(* Logix 5000 project; controller Carpenter_Meter_SCP vendor 1 type 14 code 217 rev 31.11; software revision 31.01; part 3 of 7 *)

VAR_GLOBAL   (* controller tags *)
   AI_8800 : REAL := 0.44444445;   // Meter Skid MS8800 Oil Quality BS&W (%)
   AI_8840 : REAL;   // Meter Skid MS8840 Oil Quality BS&W (%)
   alarm_co : BOOL[32];
   Alarm_horn_req : BOOL;   // Alarm Horn Request
   alarm_horn_req_tmr : TIMER := (PRE := 1000);   // Alarm Horn Request Timer
   AlwaysOff : BOOL;   // Always Off Bit
   CAR100_Flowpath : BOOL;   // Carpenter MLV CAR100 Flow Path (1=OK)
   CAR100_HB_Fail : TGE_Alarm := (Enabled := 1, AlmInputState := 1, AlmExists := 1, InAlmAct := 1, InAlmHMI := 1, DelayTimerPRE := 30.0, DelayTimerACC := 29.999, Priority := 4);   // Carpenter MLV CAR100 Heartbeat Fail Alarm
   CAR100_HB_Prev : DINT;   // MLV CAR100 Previous Heartbeat
   CAR100_High_Pressure_SD : BOOL;   // Carpenter MLV CAR100 High Pressure Shutdown Status
   Carpenter_ISD_Command : BOOL;   // Carpenter/Hereford ISD Command from OCC (Through Pawnee)
   Carpenter_Status_Pawnee : DINT[50] := ([0] := 1144740586, [2] := -1072685029);   // Carpenter Status to Pawnee
   Carpenter_to_Pawnee_OK : BOOL := 1;   // Carpenter to Pawnee Flow Path Permissive
   CC_Cust1_Flow_Permissive : BOOL := 1;   // Customer #1 (MS8800) Flow Permissive to OCC
   CC_Cust1_Hi_WIOM : BOOL;   // Customer #1 High Water % Alarm to OCC
   CC_Cust1_Pump_Running : BOOL := 1;   // Customer #1 (MS8800) Pump Running Status to OCC
   CC_Cust1_Ready : BOOL := 1;   // Customer #1 (MS8800) Ready Status to OCC
   CC_Cust1_Shutin_Timer : REAL := 30.0;   // Customer #1 Shutin Reset Time Left to OCC
   CC_Cust1_Shutin_Timer1 : DINT := 30;   // Customer #1 Shutin Reset Time Left to OCC
   CC_Cust1_WIOM_Shutin : BOOL;   // Customer #1 Shutin Due to High High Water in Oil Monitor Alarm to OCC
   CC_Cust2_Flow_Permissive : BOOL;   // Customer #2 (MS8810) Flow Permissive to OCC
   CC_Cust3_Flow_Permissive : BOOL;   // Customer #3 (MS8820) Flow Permissive to OCC
   CC_Cust4_Flow_Permissive : BOOL;   // Customer #4 (MS8830) Flow Permissive to OCC
   CC_Cust5_Flow_Permissive : BOOL := 1;   // Customer #5 (MS8840) Flow Permissive to OCC
   CC_Cust5_Pump_Running : BOOL;   // Customer #5 (MS8840) Pump Running Status to OCC
   CC_Cust5_Ready : BOOL := 1;   // Customer #5 (MS8840) Ready Status to OCC
   CC_Hererford_Flow_Path : BOOL;   // Flow Path to Hereford
   CC_HI_8800 : BOOL;   // Meter Skid MS-8800 Intrusion Deactivate Switch to OCC
   CC_HI_8840 : BOOL;   // Meter Skid MS-8840 Intrusion Deactivate Switch to OCC
   CC_MS8800_Biocide_Flow : REAL;   // Meter Skid MS-8800 Biocide Flow Rate
   CC_MS8800_Biocide_Flow_SP : REAL := 3.7771018;   // Meter Skid MS-8800 Biocide Flow Rate Setpoint
   CC_MS8800_CustPress : OCC_Analog := (scaled := 70.41581);   // Meter Skid MS-8800 Customer Inlet Pressure to OCC
   CC_MS8810_CustPress : OCC_Analog;   // Meter Skid MS-8810 Customer Inlet Pressure to OCC
   CC_MS8820_CustPress : OCC_Analog;   // Meter Skid MS-8820 Customer Inlet Pressure to OCC
   CC_MS8830_CustPress : OCC_Analog;   // Meter Skid MS-8830 Customer Inlet Pressure to OCC
   CC_MS8840_Biocide_Flow : REAL;   // Meter Skid MS-8800 Biocide Flow Rate
   CC_MS8840_Biocide_Flow_SP : REAL := 1.3565929;   // Meter Skid MS-8800 Biocide Flow Rate Setpoint
   CC_MS8840_CustPress : OCC_Analog := (scaled := 158.50713);   // Meter Skid MS-8840 Customer Inlet Pressure to OCC
   CC_OCC_HB : DINT := 12;   // Heartbeat from OCC to SCP
   CC_Pawnee_Flow_Path : BOOL := 1;   // Flow Path to Pawnee
   CC_PI_1101 : OCC_Analog;   // Station Discharge Pressure to OCC
   CC_PV_0001 : OCC_CV := (Pos := 100.0738, PosCmd := 100.0);   // PV-0001
   CC_PV_0001_Flow_SP : DINT := 1000;   // Meter Skid MS8800 Inlet Control Valve Flow Setpoint
   CC_PV_0001_Press_SP : DINT := 5;   // Meter Skid MS8800 Inlet Control Valve Press Setpoint
   CC_PV_0041 : OCC_CV := (Pos := 32.79953, PosCmd := 33.05351);   // PV-0041
   CC_PV_0041_Flow_SP : DINT := 500;   // Meter Skid MS8840 Inlet Control Valve Flow Setpoint
   CC_PV_0041_Press_SP : DINT := 120;   // Meter Skid MS8800 Inlet Control Valve Press Setpoint
   CC_SCP_HB : DINT := 1658;   // Heartbeat from SCP to OCC
   CC_STA_Stop : BOOL;   // Station Stop Request Command from OCC
   CC_XA_0020A : BOOL;   // SCP Main Panel 24VDC Fail to OCC
   CC_XA_0021A : BOOL;   // FGP Main Panel 24VDC Fail to OCC
   CC_XI_0001 : BOOL;   // QA Building Intrusion Deactivate Switch to OCC
   CC_XI_0001A : BOOL := 1;   // QA Building Intrusion Switch to OCC
   CC_XI_0011A : BOOL := 1;   // PDC Building Intrusion Switch to OCC
   CC_XI_0011B : BOOL := 1;   // PDC Building Intrusion Deactivate Switch to OCC
   CC_XI_0020 : BOOL;   // SCP Main PLC 24VDC Failure to OCC
   CC_XI_0021 : BOOL;   // FGP Main PLC 24VDC Failure to OCC
   CC_XI_8800 : BOOL;   // Meter Skid MS-8800 Intrusion Switch to OCC
   CC_XI_8800A : BOOL;   // MS8800 SCP 24VDC Failure to OCC
   CC_XI_8800B : BOOL;   // MS8800 FGP 24VDC Failure to OCC
   CC_XI_8840 : BOOL;   // Meter Skid MS-8840 Intrusion Switch to OCC
   CC_XI_8840A : BOOL;   // MS8840 SCP 24VDC Failure to OCC
   CC_XI_8840B : BOOL;   // MS8840 FGP 24VDC Failure to OCC
   CC_YI_6000 : BOOL;   // UPS-6000 Utility Power Loss to OCC
   CC_YI_6001 : BOOL;   // UPS-6000 Fault
   CC_ZI_1100A : BOOL;   // Pig Launched Pig Sig to OCC
   CC_ZI_1100B : BOOL;   // Pig Station Depart Pig Sig to OCC
   CCS_AI_0001 : OCC_Analog := (scaled := 0.024822354);   // QA Building Gas Detector to OCC (AIT-0001)
   CCS_AI_8800A : OCC_Analog := (scaled := 0.18368065);   // Meter Skid MS-8800 Gas Detector #1 (AIT-8800A)
   CCS_AI_8800B : OCC_Analog := (scaled := 0.21929741);   // Meter Skid MS-8800 Gas Detector #2 (AIT-8800B)
   CCS_AI_8840A : OCC_Analog := (scaled := 0.25642216);   // Meter Skid MS-8840 Gas Detector #1 (AIT-8840A)
   CCS_AI_8840B : OCC_Analog := (scaled := 0.22641718);   // Meter Skid MS-8840 Gas Detector #2 (AIT-8840B)
   CCS_ESD_Active : BOOL;   // Station ESD Active to OCC
   CCS_ESD_OCC : BOOL;   // Station ESD Command from OCC
   CCS_FGP_Deactivate : BOOL;   // Fire and Gas Deactivated Status to OCC
   CCS_HI_0011A : BOOL;   // PDC ESD Pushbutton to OCC
   CCS_HI_0017 : BOOL;   // PDC Building PLC Panel ESD Pushbutton to OCC
   CCS_HI_0112A : BOOL;   // QA Building ESD Pushbutton #1 to OCC
   CCS_HI_0112B : BOOL;   // QA Building ESD Pushbutton #2 to OCC
   CCS_HI_0113 : BOOL;   // South Gate ESD Pushbutton to OCC
   CCS_HI_0114 : BOOL;   // North Gate ESD Pushbutton to OCC
   CCS_HI_0115 : BOOL;   // Site ESD Pushbutton #3 to OCC - Currently Unused
   CCS_HI_8800A : BOOL;   // Meter Skid MS-8800 ESD Pushbutton #1 to OCC
   CCS_HI_8800B : BOOL;   // Meter Skid MS-8800 ESD Pushbutton #2 to OCC
   CCS_HI_8840A : BOOL;   // Meter Skid MS-8840 ESD Pushbutton #1 to OCC
   CCS_HI_8840B : BOOL;   // Meter Skid MS-8840 ESD Pushbutton #1 to OCC
   CCS_LAH_3000 : BOOL;   // Sump Tank TU-3000 Leak Detection Switch to OCC
   CCS_LAH_3000_inhibit : BOOL;   // Sump Tank TU-3000 Leak Detection Switch Inhibited to OCC
   CCS_LAH_3100 : BOOL;   // Sump Tank TU-3100 Leak Detection Switch to OCC
   CCS_LAH_3100_inhibit : BOOL;   // Sump Tank TU-3100 Leak Detection Switch Inhibited to OCC
   CCS_LAHH_3000 : BOOL;   // Sump Tank TU-3000 HiHi Level Switch to OCC
   CCS_LAHH_3000_inhibit : BOOL;   // Sump Tank TU-3000 HiHi Level Switch Inhibited to OCC
   CCS_LAHH_3100 : BOOL;   // Sump Tank TU-3100 HiHi Level Switch to OCC
   CCS_LAHH_3100_inhibit : BOOL;   // Sump Tank TU-3100 HiHi Level Switch inhibited to OCC
   CCS_LI_3000 : OCC_Analog;   // Sump Tank TU-3000 Level to OCC
   CCS_LI_3100 : OCC_Analog := (scaled := 27.158325);   // Sump Tank TU-3000 Level to OCC
   CCS_TI_8010 : OCC_Analog := (scaled := -50.0);   // PDC Building Temperature (TIT-8010)
   CCS_XI_0029A : BOOL;   // QA Building Smoke Detector #1 to OCC
   CCS_XI_0029A_Inhibit : BOOL;   // QA Building Smoke Detector #1 Inhibit to OCC
   CCS_XI_0029B : BOOL;   // QA Building Smoke Detector #2 to OCC
   CCS_XI_0029B_Inhibit : BOOL;   // QA Building Smoke Detector #2 Inhibit to OCC
   CCS_XV_0001 : BaseVLVLiquid := (chg_tmr.PRE := 180000, Close_Req_Tmr.PRE := 20000, Expected := 1, Last_Pos := 1, Open_Req_Tmr.PRE := 20000, Opn_Sts := 1, Startup_bit := 1, Startup_tmr.PRE := 120000, remote := 1, OOP_alm.sta_attended := 1, OOP_alm.alm_tmr_pre := 180000, status := 1);   // XV-0001 OCC
   CCS_XV_0041 : BaseVLVLiquid := (chg_tmr.PRE := 180000, Close_Req_Tmr.PRE := 20000, Expected := 1, Last_Pos := 1, Open_Req_Tmr.PRE := 20000, Opn_Sts := 1, Startup_bit := 1, Startup_tmr.PRE := 120000, remote := 1, OOP_alm.sta_attended := 1, OOP_alm.alm_tmr_pre := 180000, status := 1);   // XV-0041 OCC
   CCS_XV_1100 : BaseVLVLiquid := (chg_tmr.PRE := 180000, Close_Req_Tmr.PRE := 20000, Cls_Sts := 1, Open_Req_Tmr.PRE := 20000, Startup_bit := 1, Startup_tmr.PRE := 120000, remote := 1, OOP_alm.sta_attended := 1, OOP_alm.alm_tmr_pre := 180000, status := 2);   // XV-1100 OCC
   CCS_XV_1101 : BaseVLVLiquid := (chg_tmr.PRE := 180000, Close_Req_Tmr.PRE := 20000, Expected := 1, Last_Pos := 1, Open_Req_Tmr.PRE := 20000, Opn_Sts := 1, Startup_bit := 1, Startup_tmr.PRE := 120000, remote := 1, OOP_alm.sta_attended := 1, OOP_alm.alm_tmr_pre := 180000, status := 1);   // XV-1101 OCC
   CCS_YI_0022A : BOOL;   // PDC Smoke Detector to OCC
   CCS_YI_0022A_Inhibit : BOOL;   // PDC Smoke Detector Inhibit to OCC
   cmd_reset_tmr : TIMER[8] := ([0].PRE := 2000, [1].PRE := 2000, [2].PRE := 2000);   // General Use HMI Command Reset Timer
   Cust1_WIOM_Alarm : BOOL;   // Customer 1 WIOM Alarm
   Cust1_WIOM_High_Tmr : TIMER := (PRE := 900000, ACC := 82173, EN := 1, TT := 1);   // Customer 1 Water in Oil Monitor Alarm Timer
   Cust1_WIOM_Reset : BOOL;   // Customer 1 WIOM Reset Lockout from HMI
   Cust1_WIOM_Reset_Tmr : TIMER := (PRE := 1800000);   // Customer 1 Reset Timer for a WIOM Shutin
   Customer1_Flowpath_OK : BOOL := 1;   // Customer #1 Flowpath Permissive (1 = OK)
   Customer1_Pump_Status : BOOL := 1;   // Customer #1 Pump Running Status
   Customer1_Ready_Status : BOOL := 1;   // Customer #1 Ready Status
   Customer2_Flowpath_OK : BOOL;   // Customer #1 Flowpath Permissive (1 = OK)
   Customer3_Flowpath_OK : BOOL;   // Customer #3 Flowpath Permissive (1 = OK)
   Customer4_Flowpath_OK : BOOL;   // Customer #4 Flowpath Permissive (1 = OK)
   Customer4_HB : DINT;
   Customer5_Flowpath_OK : BOOL := 1;   // Customer #5 Flowpath Permissive (1 = OK)
   Customer5_Ready_Status : BOOL := 1;   // Customer #4 Ready Status
   DI_8800 : REAL := 35.538742;   // Meter Skid MS8800 Density (API)
   DI_8800_Batch : REAL := 35.5;   // Meter Skid MS8800 Current Batch Density (API)
   DI_8800_Live : REAL := 36.08286;   // Meter Skid MS8800 Live Observed Density (API)
   DI_8800_PrevBatch : REAL := 35.3;   // Meter Skid MS8800 Previous Batch Density (API)
   DI_8840 : REAL := 34.859913;   // Meter Skid MS8840 Density (API)
   DI_8840_Batch : REAL := 34.9;   // Meter Skid MS8840 Current Batch Density (API)
   DI_8840_Live : REAL := 34.490906;   // Meter Skid MS8840 Indicated Volume (Raw) (BBL/HR)
   DI_8840_PrevBatch : REAL := 35.2;   // Meter Skid MS8840 Previous Batch Density (API)
   fgp_deactivate_keysw : BOOL;   // Fire and Gas System Deactivated through Key Switch
   FGP_ESD : TGE_Alarm := (Enabled := 1, AlmExists := 1);   // ESD Shutdown from FGP (HS-0020A)
   FGP_Fire_Det : TGE_Alarm := (Enabled := 1, AlmExists := 1);   // Fire Shutdown from FGP (YSHH-0022)
   FGP_Gas_Det : TGE_Alarm := (Enabled := 1, AlmExists := 1);   // Hi Gas Shutdown from FGP (ASHH-0021)
   FGP_HB_Fail_Alm : TGE_Alarm := (Enabled := 1, AlmExists := 1);   // FGP Heartbeat Failure Alarm
   fgp_panel_reset : BOOL;   // FGP Panel Reset Pushbutton
   FGP_Produced : BasProdCons := (integer[1] := 6, integer[2] := 5, integer[3] := 5, integer[7] := 5, float[30] := 21829.0);   // FGP Produced Data
   FGP_SCADA : BasProdCons := (bit[31] := 1, bit[34] := 1, float[0] := 0.15720427, float[1] := 0.20538867, float[2] := 0.20030737, float[3] := 0.27327836, float[4] := 0.22177398, float[5] := -50.0);
   FI_8800 : REAL := 749.4378;   // Meter Skid MS-8800 Flow Rate in GSV from EFM
   FI_8800_Batch : REAL := 122.67;   // Meter Skid MS8800 Current Batch Volume in GSV (BBL)
   FI_8800_PrevBatch : REAL := 15693.27;   // Meter Skid MS8800 Pervious Batch Volume in GSV (BBL)
   FI_8800_Raw : REAL := 739.0667;   // Meter Skid MS8800 Indicated Volume (Raw) (BBL/HR)
   FI_8840 : REAL := 364.02893;   // Meter Skid MS-8840 Flow Rate from EFM
   FI_8840_Batch : REAL := 43.56;   // Meter Skid MS8840 Current Batch Volume in GSV (BBL)
   FI_8840_PrevBatch : REAL := 4837.04;   // Meter Skid MS8840 Pervious Batch Volume in GSV (BBL)
   FI_8840_Raw : REAL := 371.8956;   // Meter Skid MS8840 Indicated Volume (Raw) (BBL/HR)
   FQI_8800_DriveGain : REAL := 3.6537004;   // Meter Skid MS8800 Drive Gain (%)
   FQI_8800_Factor : REAL;   // Meter Skid MS8800 Meter Factor
   FQI_8800_LastMonth : REAL;   // Meter Skid MS8800 Gross Standard Volume Last Month (BBL)
   FQI_8800_MassFlow : REAL := 3645.5835;   // Meter Skid MS8800 Coriolis Mass Flow Rate (lb/min)
   FQI_8800_MassTotal : REAL := 774424400.0;   // Meter Skid MS8800 Coriolis Mass Totalizer (lb)
   FQI_8800_ThisMonth : REAL;   // Meter Skid MS8800 Gross Standard Volume This Month (BBL)
   FQI_8800_Today : REAL;   // Meter Skid MS8800 Gross Standard Volume Today (BBL)
   FQI_8800_Total : REAL;   // Meter Skid MS8800 Gross Standard Volume Total (BBL)
   FQI_8800_Yesterday : REAL;   // Meter Skid MS8800 Gross Standard Volume Yesterday (BBL)
   FQI_8840_DriveGain : REAL := 7.312943;   // Meter Skid MS8840 Drive Gain (%)
   FQI_8840_Factor : REAL;   // Meter Skid MS8840 Meter Factor
   FQI_8840_LastMonth : REAL;   // Meter Skid MS8840 Gross Standard Volume Last Month (BBL)
   FQI_8840_MassFlow : REAL := 1854.8619;   // Meter Skid MS8840 Coriolis Mass Flow Rate (lb/min)
   FQI_8840_MassTotal : REAL := 46132996.0;   // Meter Skid MS8840 Coriolis Mass Totalizer (lb)
   FQI_8840_ThisMonth : REAL;   // Meter Skid MS8840 Gross Standard Volume This Month (BBL)
   FQI_8840_Today : REAL;   // Meter Skid MS8840 Gross Standard Volume Today (BBL)
   FQI_8840_Total : REAL;   // Meter Skid MS8840 Gross Standard Volume Total (BBL)
   FQI_8840_Yesterday : REAL;   // Meter Skid MS8840 Gross Standard Volume Yesterday (BBL)
   hb_fail_FGP : BOOL;   // FGP Heartbeat Fail
   hb_fail_scada : BOOL;   // SCADA HB Failure
   hb_FGP : DINT := 22489;   // FGP Heartbeat
   hb_fgp_old : DINT := 22669;   // Old OCC HB for diagnostic purposes
   hb_timer_FGP : TIMER := (PRE := 600000, ACC := 15, EN := 1, TT := 1);   // FGP HB Timer
   hb_timer_scada : TIMER := (PRE := 600000, ACC := 841, EN := 1, TT := 1);   // SCADA HB Timer
   Hereford_Flowpath : BOOL := 1;   // Pawnee Terminal Flow Path (1=OK)
   Hereford_HB_Fail : TGE_Alarm := (Enabled := 1, AlmInputState := 1, AlmExists := 1, DelayTimerPRE := 30.0, DelayTimerACC := 1.527, Priority := 4);   // Hereford Heartbeat Fail Alarm
   Hereford_HB_Prev : DINT := 52;   // Hereford Previous Heartbeat
   Hereford_High_Pressure_SD : BOOL;   // Hereford High Pressure Shutdown Status
   Hereford_Msg1 : MESSAGE;
        MessageParameters(ServiceCode := 16#004c, LocalElement := Hereford_Status[0], ...)
   Hereford_OCC_HB_FAIL : BOOL;   // Pawnee High Pressure Shutdown Status
   Hereford_Status : DINT[50] := ([0] := 52, [1] := 1);   // Hereford Status Tags
   HRF100_Flowpath : BOOL := 1;   // Hereford MLV HRF100 Flow Path (1=OK)
   HRF100_HB_Fail : TGE_Alarm := (Enabled := 1, AlmInputState := 1, AlmExists := 1, DelayTimerPRE := 30.0, DelayTimerACC := 1.879);   // Hereford MLV HRF100 Heartbeat Fail Alarm
   HRF100_HB_Prev : DINT := 16;   // Hereford MLV HRF100 Previous Heartbeat
   HRF100_High_Pressure_SD : BOOL;   // Hereford MLV HRF100 High Pressure Shutdown Status
   intrusion_sys_active : BOOL;   // Intrusion System Active
   Launcher_Pig_Sig : TGE_Alarm := (Enabled := 1, AlmExists := 1);   // Launcher Pig Signal (ZS-1100A)
   Main_FGP_24VDC_Fail : TGE_Alarm := (Enabled := 1, AlmExists := 1);   // Main PLC FGP 24VDC Fail (XS-0021)
   message_timer : TIMER[10] := ([0].PRE := 5000, [0].ACC := 4855, [0].EN := 1, [0].TT := 1, [1].PRE := 2000, [1].ACC := 821, [1].EN := 1, [1].TT := 1, [2].PRE := 2000, [4].PRE := 2000);
   MLV_CAR100_Msg1 : MESSAGE;   // Carpenter MLV (CAR100) Messaging
        MessageParameters(ServiceCode := 16#004c, LocalElement := MLV_CAR100_Status[0], ...)
   MLV_CAR100_Status : DINT[50];
   MLV_HRF100_Msg1 : MESSAGE;   // Hereford MLV (HRF100) Messaging
        MessageParameters(ServiceCode := 16#004c, LocalElement := MLV_HRF100_Status[0], ...)
   MLV_HRF100_Status : DINT[50] := ([0] := 16, [1] := 1);
   mod_faultcode : DINT[10];   // PLC Module Fault Code
        [0]   // Controller Fault Code
        [1]   // SCP Main Flex I/O Fault Code
        [2]   // Meter Skid MS8800 RIO Fault Code
        [3]   // Meter Skid MS8810 RIO Fault Code
        [4]   // Meter Skid MS8820 RIO Fault Code
        [5]   // Meter Skid MS8830 RIO Fault Code
        [6]   // Meter Skid MS8840 RIO Fault Code
   mod_status : DINT[10] := ([0] := 12640, [1] := 16384, [2] := 16384, [6] := 16384, [8] := 2);   // PLC Module Status
        [0]   // Controller Module Status
        [1]   // SCP Main Flex I/O Module Status
        [2]   // Meter Skid MS8800 RIO Module Status
        [3]   // Meter Skid MS8810 RIO Module Status
        [4]   // Meter Skid MS8820 RIO Module Status
        [5]   // Meter Skid MS8830 RIO Module Status
        [6]   // Meter Skid MS8840 RIO Module Status
   MS8800_Biocide_BBL_Per_Day : REAL := 0.08833598;   // MS8800 Biocide Flow Rate in BBL/Day (Based off set target of 500PPM)
   MS8800_Biocide_Flow_Fdbk : TGE_AI_UDT := (TrendTime := 1, Raw := -3.2007636e-05, HHAlm.AlmInputState := 1, HHAlm.AlmExists := 1, HAlm.AlmInputState := 1, HAlm.AlmExists := 1, LAlm.AlmInputState := 1, LAlm.AlmExists := 1, LLAlm.AlmInputState := 1, LLAlm.AlmExists := 1, ROCNegAlm.AlmExists := 1, ROCPosAlm.AlmExists := 1, MalfAlm.AlmInputState := 1, MalfAlm.AlmExists := 1);   // Meter Skid MS-8800 Biocide Injection Rate Feedback
   MS8800_Biocide_Flow_Fdbk_AOI : TGE_AI := (Raw := -2.8205577e-05);   // Meter Skid MS-8800 Biocide Injection Rate Feedback
   MS8800_Biocide_Flow_SP : REAL := 3.7771666;   // Meter Skid MS-8800 Biocide Flow Rate Gal/Day
   MS8800_Biocide_RunReq : BOOL := 1;   // Meter Skid MS8800 Biocide Run Req
   MS8800_Cust_Press : TGE_AI_UDT := (TrendTime := 1, Avg := 70.44822, EU := 70.44822, EUMax := 1500.0, Raw := 4.7514477, RawMax := 20.0, RawMin := 4.0, Percent := 4.696548, HHAlm.AlmInputState := 1, HHAlm.AlmExists := 1, HAlm.AlmInputState := 1, HAlm.AlmExists := 1, LAlm.AlmExists := 1, LLAlm.AlmExists := 1, ROCNegAlm.AlmExists := 1, ROCPosAlm.AlmExists := 1, MalfAlm.AlmExists := 1, Average.Input := 70.44822, Average.Output := 70.44822);   // Meter Skid MS-8800 Customer Inlet Pressure (Communicated from Cust)
   MS8800_Cust_Press_AOI : TGE_AI := (Raw := 4.7514477, EU := 70.44822, Avg := 70.44822);   // Meter Skid MS-8800 Customer Inlet Pressure (Communicated from Cust)
   MS8800_Customer_Inlet_Press : AnalogAlm := (mA := 4.0, sta_attended := 1, Lo_setpt := -1.0, LoLo_setpt := -1.0, Hi_setpt := 1368.0, HiHi_setpt := 1425.0);   // Meter Skid MS8800 Customer Inlet Pressure
   MS8800_CustPress : REAL;
   MS8800_EFM_Data : REAL[50] := ([0] := 736.1332, [1] := 55.73959, [2] := 67.49643, [3] := 35.54057, [4] := 123.28, [5] := 63.0, [6] := 67.3, [7] := 35.5, [8] := 15693.27, [9] := 138.0, [10] := 65.9, [11] := 35.3, [12] := 738.34155, [13] := 36.08286, [15] := 0.44444445, [16] := 31.093464, [17] := 1.6411064, [18] := 3645.5835, [19] := 774424400.0, [20] := 3.6537004);   // MS8800 EFM Data Points
        [0]   // Live GSV Rate from MS8800 EFM
        [1]   // Live Static Pressure from MS8800 EFM
        [2]   // Live Temperature from MS8800 EFM
        [3]   // Current Batch GSV Total from MS8800 EFM
        [4]   // Current Batch FWA Static Pressure from MS8800 EFM
        [5]   // Current Batch FWA Temperature from MS8800 EFM
        [6]   // Current Batch FWA Base Density from MS8800 EFM
        [7]   // Previous Batch GSV Total from MS8800 EFM
        [8]   // Previous Batch FWA Static Pressure from MS8800 EFM
        [9]   // Previous Batch FWA Temperature from MS8800 EFM
        [10]   // Previous Batch FWA Base Density from MS8800 EFM
        [11]   // Live Indicated Volume (Raw) Rate from MS8800 EFM
        [12]   // Live Observed Density from MS8800 EFM
        [13]   // GSV Accumulator Grand Total from MS8800 EFM
        [14]   // WIOM / H20 / BSW from MS8800 EFM
        [15]   // Control Valve Position Feedback from MS8800 EFM
        [16]   // Strainer Differential from MS8800 EFM
        [17]   // Coriolis Mass Rate from MS8800 EFM
        [18]   // Coriolis Mass Totalizer from MS8800 EFM
        [19]   // Drive Gain from MS8800 EFM
        [20]   // Meter Factor from MS8800 EFM
        [21]   // Today GSV Total from MS8800 EFM
        [22]   // Yesterday GSV Total from MS8800 EFM
        [23]   // This Month GSV Total from MS8800 EFM
        [24]   // Last Month GSV Total from MS8800 EFM
   MS8800_FGP_24VDC_Fail : TGE_Alarm := (Enabled := 1, AlmExists := 1, DelayTimerPRE := 5.0, DelayTimerACC := 4.999);   // Meter Skid MS-8800 FGP 24VDC Fail (XS-8800B)
   MS8800_Flow_Control : PID := (CTL := -2147446144, EN := 1, INI := 1, OLH := 1, DVPA := 1, PVHA := 1, SP := 1000.0, KP := 0.0025, KI := 0.001, MAXS := 5000.0, DB := 7.0, SO := 100.0, MAXO := 100.0, UPD := 0.2, PV := 750.19684, ERR := 249.80316, OUT := 100.0, MAXI := 5000.0, MAXCV := 100.0, MAXTIE := 4095.0, DATA[0] := 99.99973, DATA[1] := -240.06299, DATA[2] := 750.19684, DATA[3] := 249.80316, DATA[4] := 1000.0, DATA[5] := 0.02, DATA[6] := 1.0, DATA[7] := 3.2, DATA[8] := 0.0025, DATA[9] := 0.001, DATA[11] := 0.0025, DATA[12] := 0.001, DATA[15] := 1.0, DATA[16] := 0.024420025);   // Meter Skid MS8800 Flow Rate P&ID
   MS8800_Inlet_Press : TGE_AI_UDT := (HHAlm.AlmExists := 1, HAlm.AlmExists := 1, LAlm.AlmExists := 1, LLAlm.AlmExists := 1, ROCNegAlm.AlmExists := 1, ROCPosAlm.AlmExists := 1, MalfAlm.AlmExists := 1);   // Meter Skid MS-8800 Inlet Pressure
   MS8800_Inlet_Press_AOI : TGE_AI;   // Meter Skid MS-8800 Inlet Pressure
   MS8800_Inlet_Press_Control : PID := (CTL := -2113891712, EN := 1, CA := 1, INI := 1, OLH := 1, DVPA := 1, PVHA := 1, SP := 5.0, KP := 0.2, KI := 0.05, MAXS := 1500.0, DB := 2.0, SO := 100.0, MAXO := 100.0, UPD := 0.2, PV := 70.54263, ERR := 65.54263, OUT := 100.0, MAXI := 1500.0, MAXCV := 100.0, MAXTIE := 4095.0, DATA[0] := 99.8426, DATA[1] := 75.245476, DATA[2] := 70.54263, DATA[3] := 65.54263, DATA[4] := 5.0, DATA[5] := 0.06666667, DATA[6] := 1.0, DATA[7] := 1.6, DATA[8] := 0.2, DATA[9] := 0.05, DATA[11] := 0.2, DATA[12] := 0.05, DATA[15] := 1.0, DATA[16] := 0.024420025);   // Meter Skid MS8800 Customer Inlet Pressure P&ID
   MS8800_Intrusion : IntrusionAlm := (sta_attended := 1, sw_input := 7);   // Meter Skid MS-8800 Intrusion #1 Alarm
   MS8800_OilFlow_BBL_Per_Day : REAL := 17986.508;   // Meter Skid MS-8800 Oil Flow Rate in BBL/Day
   MS8800_PCV_Pos : TGE_AI_UDT := (TrendTime := 1, Avg := 100.0739, EU := 100.0739, EUMax := 100.0, Raw := 100.0739, RawMax := 100.0, Percent := 100.0739, HHAlm.AlmInputState := 1, HHAlm.AlmExists := 1, HAlm.AlmInputState := 1, HAlm.AlmExists := 1, LAlm.AlmExists := 1, LLAlm.AlmExists := 1, ROCNegAlm.AlmExists := 1, ROCPosAlm.AlmExists := 1, MalfAlm.AlmExists := 1, Average.Input := 100.0739, Average.Output := 100.0739);   // Meter Skid MS-8800 Pressure Control Valve - Position Feedback (PCV-0001)
   MS8800_PCV_Pos_AOI : TGE_AI := (Raw := 100.07354, EU := 100.07354, Avg := 100.07354);   // Meter Skid MS-8800 Pressure Control Valve - Position Feedback (PCV-0001)
   MS8800_RIO_Fail : TGE_Alarm := (AlmInputState := 1, AlmExists := 1);   // MS8800 RIO Failure
   MS8800_WaterFlow_BBL_Per_Day : REAL := 176.67195;   // MS8800 Water Flow Rate in BBL/Day (Based off 1% oil in water)
   MS8800_WIOM_Alarm : AnalogAlm := (Input := 0.44566545, mA := 4.0, sta_attended := 1, Hi_setpt := 1.5, HiHi_setpt := 1.7, Hi_tmr_pre := 300000, HiHi_tmr_pre := 900000);   // MS8800 Water In Oil Monitor Alarm (Setpoint Dictated by Tarrif)
   MS8810_RIO_Fail : TGE_Alarm := (AlmExists := 1);   // MS8810 RIO Failure
   MS8840_Biocide_BBL_Per_Day : REAL := 0.044638067;   // MS8840 Biocide Flow Rate in BBL/Day (Based off set target of 500PPM)
   MS8840_Biocide_Flow_Fdbk : TGE_AI_UDT := (TrendTime := 1, Raw := 0.00016698558, HHAlm.AlmInputState := 1, HHAlm.AlmExists := 1, HAlm.AlmInputState := 1, HAlm.AlmExists := 1, LAlm.AlmInputState := 1, LAlm.AlmExists := 1, LLAlm.AlmInputState := 1, LLAlm.AlmExists := 1, ROCNegAlm.AlmExists := 1, ROCPosAlm.AlmExists := 1, MalfAlm.AlmInputState := 1, MalfAlm.AlmExists := 1);   // Meter Skid MS-8840 Biocide Injection Rate Feedback
   MS8840_Biocide_Flow_Fdbk_AOI : TGE_AI := (Raw := 0.00015556542);   // Meter Skid MS-8840 Biocide Injection Rate Feedback
   MS8840_Biocide_Flow_SP : REAL := 1.8475137;   // Meter Skid MS-8840 Biocide Flow Rate Gal/Day
   MS8840_Biocide_RunReq : BOOL := 1;   // Meter Skid MS8840 Biocide Run Req
   MS8840_Cust_Press : TGE_AI_UDT := (TrendTime := 1, Avg := 151.95697, EU := 151.95697, EUMax := 1650.0, Raw := 5.473522, RawMax := 20.0, RawMin := 4.0, Percent := 9.209514, HHAlm.AlmInputState := 1, HHAlm.AlmExists := 1, HAlm.AlmInputState := 1, HAlm.AlmExists := 1, LAlm.AlmExists := 1, LLAlm.AlmExists := 1, ROCNegAlm.AlmExists := 1, ROCPosAlm.AlmExists := 1, MalfAlm.AlmExists := 1, Average.Input := 151.95697, Average.Output := 151.95697);   // Meter Skid MS-8840 Customer Inlet Pressure (Communicated from Cust)
   MS8840_Cust_Press_AOI : TGE_AI := (Raw := 5.469001, EU := 151.4907, Avg := 151.4907);   // Meter Skid MS-8840 Customer Inlet Pressure (Communicated from Cust)
   MS8840_Customer_Inlet_Press : AnalogAlm := (mA := 4.0, sta_attended := 1, Lo_setpt := -1.0, LoLo_setpt := -1.0, Hi_setpt := 1368.0, HiHi_setpt := 1425.0);   // Meter Skid MS8840 Customer Inlet Pressure
   MS8840_CustPress : REAL;   // Meter Skid MS8840 Customer Inlet Pressure from Customer
   MS8840_EFM_Data : REAL[50] := ([0] := 371.9839, [1] := 110.6033, [2] := 56.4323, [3] := 34.859913, [4] := 43.56, [5] := 89.0, [6] := 56.4, [7] := 34.9, [8] := 4837.04, [9] := 124.0, [10] := 56.2, [11] := 35.2, [12] := 371.15622, [13] := 34.487686, [16] := 23.901098, [17] := 1.2, [18] := 1852.3253, [19] := 46132870.0, [20] := 7.3661847);   // MS8840 EFM Data Points
   MS8840_EFM_DINTs : DINT[10] := ([0] := 17955, [1] := 1, [2] := 144, [3] := 34, [5] := 1);   // MS8840 EFM DINT Points
        [5].1   // MS8840 EFM DINT Points
   MS8840_EFM_ReadBools : BOOL[32];   // MS8840 EFM Read Bools
   MS8840_EFM_WriteBools : BOOL[32];   // MS8840 EFM Writen Bools
   MS8840_FGP_24VDC_Fail : TGE_Alarm := (Enabled := 1, AlmExists := 1);   // Meter Skid MS-8840 FGP 24VDC Fail (XS-8840B)
   MS8840_Flow_Control : PID := (CTL := 37504, INI := 1, OLH := 1, DVPA := 1, PVHA := 1, SP := 500.0, KP := 0.1, KI := 1.0, MAXS := 5000.0, DB := 7.5, SO := 100.0, MAXO := 100.0, UPD := 0.2, PV := 368.7331, ERR := 131.2669, OUT := 100.0, MAXI := 5000.0, MAXCV := 100.0, MAXTIE := 4095.0, DATA[0] := 99.77896, DATA[1] := -117.99459, DATA[2] := 368.7331, DATA[3] := 131.2669, DATA[4] := 500.0, DATA[5] := 0.02, DATA[6] := 1.0, DATA[7] := 3.2, DATA[8] := 0.1, DATA[9] := 1.0, DATA[11] := 0.1, DATA[12] := 1.0, DATA[15] := 1.0, DATA[16] := 0.024420025);   // Meter Skid MS8840 Flow Rate P&ID
   MS8840_Inlet_Press : TGE_AI_UDT := (HHAlm.AlmExists := 1, HAlm.AlmExists := 1, LAlm.AlmExists := 1, LLAlm.AlmExists := 1, ROCNegAlm.AlmExists := 1, ROCPosAlm.AlmExists := 1, MalfAlm.AlmExists := 1);   // Meter Skid MS-8840 Inlet Pressure (From EFM)
   MS8840_Inlet_Press_AOI : TGE_AI;   // Meter Skid MS-8840 Inlet Pressure (From EFM)
   MS8840_Inlet_Press_Control : PID := (CTL := 43025024, CA := 1, PE := 1, NOZC := 1, INI := 1, DVPA := 1, PVHA := 1, SP := 120.0, KP := 0.45, KI := 0.12, MAXS := 1650.0, DB := 2.0, SO := 33.07294, MAXO := 100.0, UPD := 0.2, PV := 147.57181, ERR := 27.571808, OUT := 33.07294, MAXI := 1650.0, MAXCV := 100.0, MAXTIE := 4095.0, DATA[0] := 32.320984, DATA[1] := 143.09995, DATA[2] := 147.57181, DATA[3] := 27.571808, DATA[4] := 120.0, DATA[5] := 0.060606062, DATA[6] := 1.0, DATA[7] := 3.2, DATA[8] := 0.45, DATA[9] := 0.12, DATA[11] := 0.45, DATA[12] := 0.0625, DATA[15] := 1.0, DATA[16] := 0.024420025);   // Meter Skid MS8840 Customer Inlet Pressure P&ID
   MS8840_Intrusion : IntrusionAlm := (sta_attended := 1, sw_input := 15);   // Meter Skid MS-8840 Intrusion Alarm
   MS8840_OilFlow_BBL_Per_Day : REAL := 8797.684;   // Meter Skid MS-8840 Oil Flow Rate in BBL/Day
   MS8840_PCV_Pos : TGE_AI_UDT := (TrendTime := 1, Avg := 31.225883, EU := 31.225883, EUMax := 100.0, Raw := 8.996141, RawMax := 20.0, RawMin := 4.0, Percent := 31.225883, HHAlm.AlmInputState := 1, HHAlm.AlmExists := 1, HAlm.AlmInputState := 1, HAlm.AlmExists := 1, LAlm.AlmExists := 1, LLAlm.AlmExists := 1, ROCNegAlm.AlmExists := 1, ROCPosAlm.AlmExists := 1, MalfAlm.AlmExists := 1, Average.Input := 31.225883, Average.Output := 31.225883);   // Meter Skid MS-8840 Pressure Control Valve - Position Feedback (PCV-0041)
   MS8840_PCV_Pos_AOI : TGE_AI := (Raw := 8.995548, EU := 31.222176, Avg := 31.222176);   // Meter Skid MS-8840 Pressure Control Valve - Position Feedback (PCV-0041)
   MS8840_RIO_Fail : TGE_Alarm := (AlmInputState := 1, AlmExists := 1);   // MS8840 RIO Failure
   MS8840_WaterFlow_BBL_Per_Day : REAL := 89.18919;   // MS8840 Water Flow Rate in BBL/Day (Based off 1% oil in water)
   OCC_hb_old : DINT := 22;   // Old OCC HB for diagnostic purposes
   OCC_WIOM_Reset : BOOL;
   OCC_WIOM_Reset_Tmr : TIMER := (PRE := 900000, ACC := 900000, EN := 1, DN := 1);
   one_sec_tmr : TIMER := (PRE := 1000, ACC := 511, EN := 1, TT := 1);   // One Second Pulse Timer
   ons_gen_use : BOOL[64];
   ovrd_disch_press : Override := (inh_sp := 1406.0, unld1_sp := 1425.0, unldall_sp := 1435.0, stop1_sp := 1450.0, sta_stop_sp := 1465.0, priority_ww := 99);   // Discharge Pressure Override
   ovrd_esd : Override := (priority_ww := 1);   // ESD Override
   ovrd_fire : Override := (priority_ww := 2);   // Fire Override
   ovrd_gas : Override := (priority_ww := 3);   // Gas Override
   Pawnee_ESD : BOOL := 1;   // Pawnee Terminal ESD Signal (1=OK, 0 = ESD Active)
   Pawnee_Flowpath : BOOL := 1;   // Pawnee Terminal Flow Path (1=OK)
   Pawnee_HB_Fail : TGE_Alarm := (Enabled := 1, AlmInputState := 1, AlmExists := 1, DelayTimerPRE := 30.0, DelayTimerACC := 3.558, Priority := 4);   // Pawnee Heartbeat Fail Alarm
   Pawnee_HB_Prev : DINT := 22;   // Pawnee Heartbeat Previous Value
   Pawnee_High_Pressure_SD : BOOL;   // Pawnee High Pressure Shutdown Status
   Pawnee_Msg1 : MESSAGE;   // Pawnee Read Message
        MessageParameters(ServiceCode := 16#004c, LocalElement := Pawnee_Status[0], ...)
   Pawnee_Msg2 : MESSAGE;   // Pawnee Write Message
        MessageParameters(ServiceCode := 16#004d, LocalElement := Carpenter_Status_Pawnee[0], ...)
   Pawnee_OCC_HB_FAIL : BOOL;   // Pawnee OCC HB Fail
   Pawnee_Status : DINT[50] := ([0] := 22, [1] := 9);   // Pawnee Status Bits
        [1].0   // Pawnee Flowpath
        [1].1   // Pawnee High Pressure Shutdown
        [1].2   // Pawnee OCC HB Fail
   PDC_Bldg_Intrusion : IntrusionAlm := (sta_attended := 1, sw_input := -32767);   // PDC Building Intrusion Alarm
   PDI_8800 : REAL := 1.6167661;   // Meter Skid MS8800 Differential Pressure
   PDI_8840 : REAL := 1.2;   // Meter Skid MS8840 Differential Pressure
   PI_8800 : REAL := 55.28271;   // Meter Skid MS8800 Pressure (PSI)
   PI_8800_Batch : REAL := 63.0;   // Meter Skid MS8800 Current Batch Pressure (PSIG)
   PI_8800_PrevBatch : REAL := 138.0;   // Meter Skid MS8800 Previous Batch Pressure (PSIG)
   PI_8840 : REAL := 111.0603;   // Meter Skid MS8840 Pressure (PSI)
   PI_8840_Batch : REAL := 89.0;   // Meter Skid MS8840 Current Batch Pressure (PSIG)
   PI_8840_PrevBatch : REAL := 124.0;   // Meter Skid MS8840 Previous Batch Pressure (PSIG)
   PIC_0001A_Out : REAL := 100.0;   // Control Valve Output Variable Related to Inlet Pressure
   PIC_0001B_Out : REAL := 100.0;   // Control Valve Ouptut Variable related to Flow Rate
   PIC_0041A_Out : REAL := 35.36881;   // Control Valve Output Variable Related to Inlet Pressure
   PIC_0041B_Out : REAL := 100.0;   // Control Valve Ouptut Variable related to Flow Rate
   PLC_Fail : TGE_Alarm := (AlmInputState := 1, AlmExists := 1, DelayTimerPRE := 2.0, DelayTimerACC := 1.9, Priority := 1);   // SCP PLC Failure
   PlcClock : LocalDateTime := (Year := 1998, Month := 6, Day := 24, Hour := 11, Minute := 27, Second := 14, mSec := 460, uSec := 460514, HhMmSs := 112714);   // PLC Clock using Get System Variables
   PV0001_Error : REAL := 0.0741806;   // PV0001 Command vs. Feedback Error
   PV0001_Error_ABS : DINT;   // PV0001 Percent Error ABS value
   PV0001_Malf : TGE_Alarm := (Enabled := 1, AlmExists := 1, DelayTimerPRE := 30.0, DelayTimerACC := 6.421);   // PV0001 Malfunction Alarm
   PV0001_Pos_Cmd : REAL := 100.0;   // PCV-0001 Position Command
   PV0041_Error : REAL := 0.40258408;   // PV0041 Command vs. Feedback Error
   PV0041_Malf : TGE_Alarm := (AlmExists := 1, DelayTimerPRE := 30.0);   // PV0041 Malfunction Alarm
   PV0041_Pos_Cmd : REAL := 35.384495;   // PCV-0041 Position Command
   pv_0001_pid_tmr : TIMER := (PRE := 200, ACC := 46, EN := 1, TT := 1);
   pv_0041_pid_tmr : TIMER := (PRE := 200, ACC := 178, EN := 1, TT := 1);
   QA_Bldg_Intrusion : IntrusionAlm := (sta_attended := 1, sw_input := 1);   // QA Building Intrusion Alarm Bit 0-7 = Bldg Int Switch Bit 15 = Deact HS
   SCADA_HB_Fail_Alm : TGE_Alarm := (Enabled := 1, AlmExists := 1);   // SCADA Hearbeat Failure Alarm
   SCP_Forces_Active : TGE_Alarm := (AlmExists := 1, DelayTimerPRE := 2.0, DelayTimerACC := 1.9, Priority := 1);   // SCP PLC Forces Active
   SCP_Main_Fail : TGE_Alarm := (AlmInputState := 1, AlmExists := 1);   // SCP Main Flex I/O Failure
   SCP_Produced : BasProdCons := (bit[10] := 1, integer[0] := 17336, integer[10] := 17); {produced}
   Sta_Stat : StaStatus := (remote := 1, attended := 1, stopping := 1, cur_ovrd_priority := 100);
   sta_stop : StaStartStop := (step_complete[0] := 1, step_complete[1] := 1, step_complete[2] := 1, step_complete[3] := 1, step_complete[4] := 1, timer[1].PRE := 180000, overall_tmr.PRE := 360000, hmi_alm_clear := 1);   // Station Stop
   sta_stop_vlv_req : BOOL;   // Station Stop Valve Close Request
   Station_Depart_Pig_Sig : TGE_Alarm := (Enabled := 1, AlmExists := 1);   // Station Departed Pig Signal (ZS-1100B)
   Station_Disch_Press : TGE_AI_UDT := (TrendTime := 1, EUMax := 1650.0, HHAlmSP := 1425.0, HAlmSP := 1368.0, Raw := 3.9500802, RawMax := 20.0, RawMin := 4.0, HHAlm.AlmExists := 1, HAlm.AlmExists := 1, LAlm.AlmInputState := 1, LAlm.AlmExists := 1, LLAlm.AlmInputState := 1, LLAlm.AlmExists := 1, ROCNegAlm.AlmExists := 1, ROCPosAlm.AlmExists := 1, MalfAlm.AlmExists := 1);   // Station Discharge Pressure - Launcher Skid (PIT-1101)
   Station_Disch_Press_AOI : TGE_AI := (Raw := 3.9508147);   // Station Discharge Pressure - Launcher Skid (PIT-1101)
   Temp_Toggle : BOOL;
   Temp_toggle2 : BOOL;
   Test : BOOL;
   Test_Bit : BOOL[32] := ([0] := 1);
   test_timer : TIMER;
   Testbits2 : DINT;   // Meter Skid MS8840 Inlet Control Valve Flow Setpoint
   TI_8800 : REAL := 67.49643;   // Meter Skid MS8800 Temperature
   TI_8800_Batch : REAL := 67.3;   // Meter Skid MS8800 Current Batch Temperature (deg F)
   TI_8800_PrevBatch : REAL := 65.9;   // Meter Skid MS8800 Previous Batch Temperature (deg F)
   TI_8840 : REAL := 56.4323;   // Meter Skid MS8840 Temperature
   TI_8840_Batch : REAL := 56.4;   // Meter Skid MS8840 Current Batch Temperature (deg F)
   TI_8840_PrevBatch : REAL := 56.2;   // Meter Skid MS8840 Previous Batch Temperature (deg F)
   TU3000_HiHi_Lvl : TGE_Alarm := (Enabled := 1, AlmExists := 1);   // Sump Tank (TU-3000) Hi Hi Level Switch (LSHH-3000)
   TU3000_Leak_Detect : TGE_Alarm := (Enabled := 1, AlmExists := 1);   // Sump Tank (TU-3000) Leak Detected (LSH-3000)
   TU3000_Level : TGE_AI_UDT := (TrendTime := 1, EUMax := 100.0, HHAlmSP := 75.0, HAlmSP := 65.0, Raw := 3.9011893, RawMax := 20.0, RawMin := 4.0, HHAlm.AlmExists := 1, HAlm.AlmExists := 1, LAlm.AlmInputState := 1, LAlm.AlmExists := 1, LLAlm.AlmInputState := 1, LLAlm.AlmExists := 1, ROCNegAlm.AlmExists := 1, ROCPosAlm.AlmExists := 1, MalfAlm.AlmExists := 1);   // Sump Tank (TU-3000) Level Transmitter (LIT-3000)
   TU3000_Level_AOI : TGE_AI := (Raw := 3.9011512);   // Sump Tank (TU-3000) Level Transmitter (LIT-3000)
   TU3100_HiHi_Lvl : TGE_Alarm := (Enabled := 1, AlmExists := 1);   // Sump Tank (TU-3100) Hi Hi Level Switch (LSHH-3100)
   TU3100_Leak_Detect : TGE_Alarm := (Enabled := 1, AlmExists := 1);   // Sump Tank (TU-3100) Leak Detected (LSH-3100)
   TU3100_Level : TGE_AI_UDT := (TrendTime := 1, Avg := 27.157562, EU := 27.157562, EUMax := 100.0, HHAlmSP := 75.0, HAlmSP := 65.0, LAlmSP := 15.0, LLAlmSP := 10.0, Raw := 8.34521, RawMax := 20.0, RawMin := 4.0, Percent := 27.157562, HHAlm.AlmExists := 1, HAlm.AlmExists := 1, LAlm.AlmExists := 1, LLAlm.AlmExists := 1, ROCNegAlm.AlmExists := 1, ROCPosAlm.AlmExists := 1, MalfAlm.AlmExists := 1, Average.Input := 27.157562, Average.Output := 27.157562);   // Sump Tank (TU-3100) Level Transmitter (LIT-3100)
   TU3100_Level_AOI : TGE_AI := (Raw := 8.3452215, EU := 27.157635, Avg := 27.157635);   // Sump Tank (TU-3100) Level Transmitter (LIT-3100)
   unit_msg_group : DINT := 2;
   UPS_Fault : TGE_Alarm := (AlmExists := 1);   // UPS-6000 Fault (YS-6001)
   UPS_Online : TGE_Alarm := (AlmExists := 1);   // UPS-6000 Loss of AC Feed (YS-6000)
   valve_failure : BOOL;   // Valve Failure Override
   valve_SD_tmr : TIMER := (PRE := 1000);   // Valve Failure Station Stop Timer
   watchdog_tmr : TIMER := (PRE := 30000, ACC := 22093, EN := 1, TT := 1);   // Watchdog Timer for Communications
   XV_0001 : BaseVLVLiquid := (chg_tmr.PRE := 180000, Close_Req_Tmr.PRE := 20000, Expected := 1, Last_Pos := 1, Open_Req_Tmr.PRE := 20000, Opn_Sts := 1, Startup_bit := 1, Startup_tmr.PRE := 120000, remote := 1, OOP_alm.sta_attended := 1, OOP_alm.alm_tmr_pre := 180000, status := 1);   // XV-0001
   XV_0001_AOI : Valve_Control := (sys_plc_perm := 1);   // XV-0001 Control
   XV_0041 : BaseVLVLiquid := (chg_tmr.PRE := 180000, Close_Req_Tmr.PRE := 20000, Expected := 1, Last_Pos := 1, Open_Req_Tmr.PRE := 20000, Opn_Sts := 1, Startup_bit := 1, Startup_tmr.PRE := 120000, remote := 1, OOP_alm.sta_attended := 1, OOP_alm.alm_tmr_pre := 180000, status := 1);   // XV-0041
   XV_0041_AOI : Valve_Control := (sys_plc_perm := 1);   // XV-0041 Control
   XV_1100 : BaseVLVLiquid := (chg_tmr.PRE := 180000, Close_Req_Tmr.PRE := 20000, Cls_Sts := 1, Open_Req_Tmr.PRE := 20000, Startup_bit := 1, Startup_tmr.PRE := 120000, remote := 1, OOP_alm.sta_attended := 1, OOP_alm.alm_tmr_pre := 180000, status := 2);   // XV-1100
   XV_1100_AOI : Valve_Control := (sys_plc_perm := 1);   // XV-1100 Control
   XV_1101 : BaseVLVLiquid := (chg_tmr.PRE := 180000, Close_Req_Tmr.PRE := 20000, Expected := 1, Last_Pos := 1, Open_Req_Tmr.PRE := 20000, Opn_Sts := 1, Startup_bit := 1, Startup_tmr.PRE := 120000, remote := 1, OOP_alm.sta_attended := 1, OOP_alm.alm_tmr_pre := 180000, status := 1);   // XV-1101
   XV_1101_AOI : Valve_Control := (sys_plc_perm := 1);   // XV-1100 Control
   ZI_8800 : REAL := 31.093464;   // Meter Skid MS8800 Back Pressure Valve Position
   ZI_8840 : REAL := 23.901098;   // Meter Skid MS8840 Back Pressure Valve Position
END_VAR

PROGRAM Alarm_Shutdown   (* main routine Alarm_Main *)

ROUTINE Alarm_Main   (* ladder *)
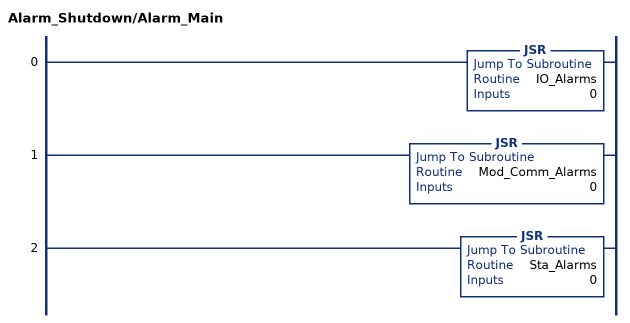
   0: JSR(IO_Alarms,0);
   1: JSR(Mod_Comm_Alarms,0);
   2: JSR(Sta_Alarms,0);
END_ROUTINE

ROUTINE IO_Alarms   (* ladder *)
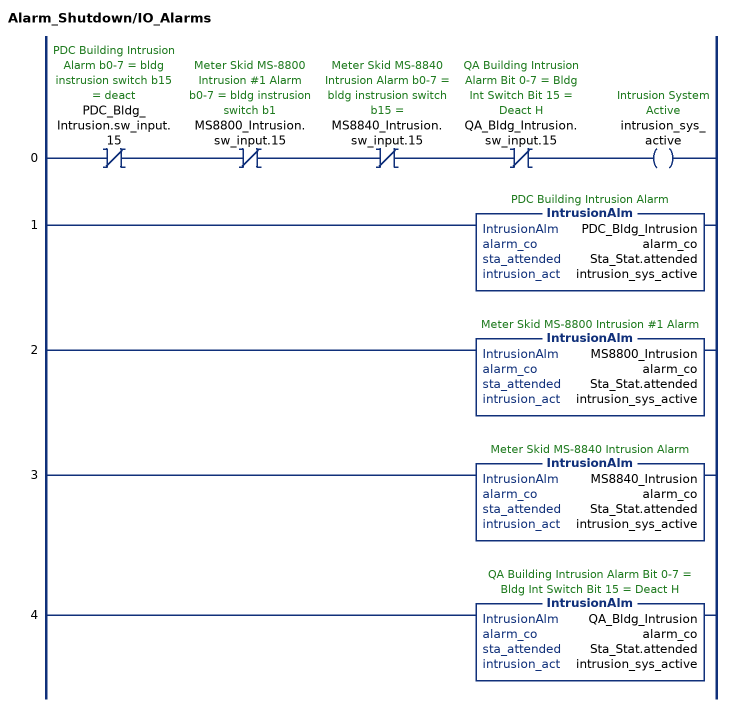
   0: XIO(PDC_Bldg_Intrusion.sw_input.15)XIO(MS8800_Intrusion.sw_input.15)XIO(MS8840_Intrusion.sw_input.15)XIO(QA_Bldg_Intrusion.sw_input.15)OTE(intrusion_sys_active);
   1: IntrusionAlm(PDC_Bldg_Intrusion,alarm_co,Sta_Stat.attended,intrusion_sys_active);
   2: IntrusionAlm(MS8800_Intrusion,alarm_co,Sta_Stat.attended,intrusion_sys_active);
   3: IntrusionAlm(MS8840_Intrusion,alarm_co,Sta_Stat.attended,intrusion_sys_active);
   4: IntrusionAlm(QA_Bldg_Intrusion,alarm_co,Sta_Stat.attended,intrusion_sys_active);
END_ROUTINE

ROUTINE Mod_Comm_Alarms   (* ladder *)
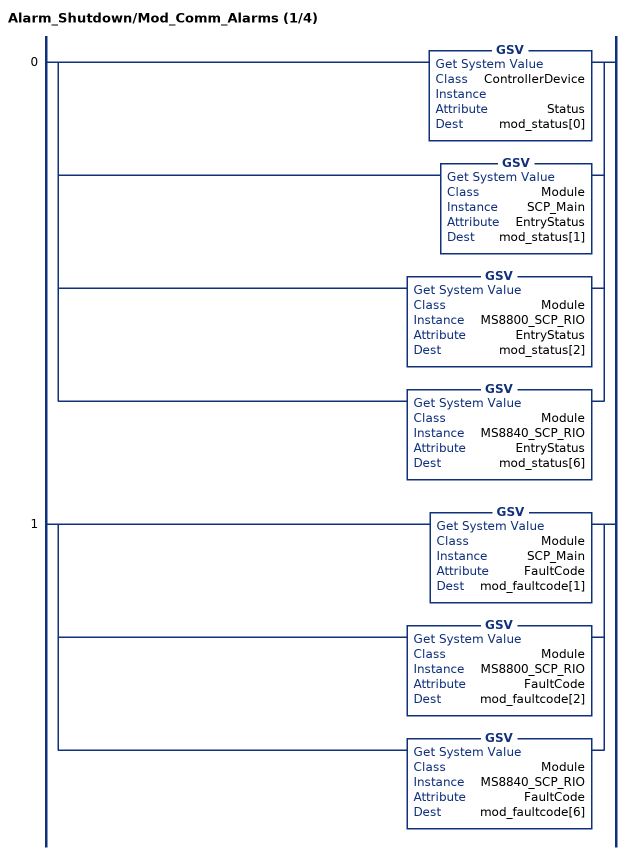
   0: [GSV(ControllerDevice,,Status,mod_status[0]) ,GSV(Module,SCP_Main,EntryStatus,mod_status[1]) ,GSV(Module,MS8800_SCP_RIO,EntryStatus,mod_status[2]) ,GSV(Module,MS8840_SCP_RIO,EntryStatus,mod_status[6]) ];
   1: [GSV(Module,SCP_Main,FaultCode,mod_faultcode[1]) ,GSV(Module,MS8800_SCP_RIO,FaultCode,mod_faultcode[2]) ,GSV(Module,MS8840_SCP_RIO,FaultCode,mod_faultcode[6]) ];
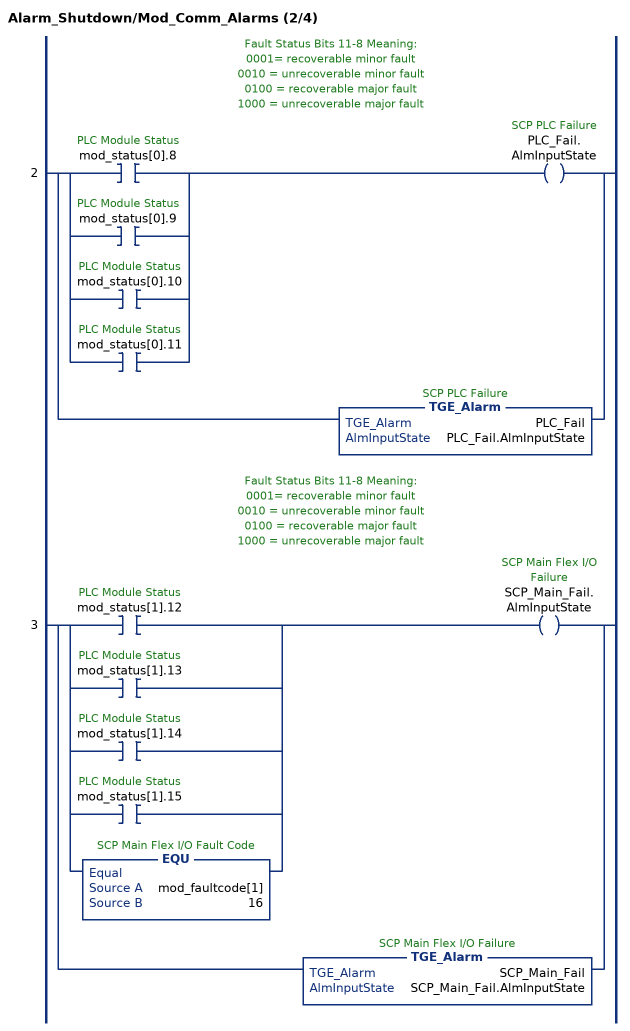
   // Fault Status Bits 11-8 Meaning:
   // 0001= recoverable minor fault
   // 0010 = unrecoverable minor fault
   // 0100 = recoverable major fault
   // 1000 = unrecoverable major fault
   2: [[XIC(mod_status[0].8) ,XIC(mod_status[0].9) ,XIC(mod_status[0].10) ,XIC(mod_status[0].11) ] OTE(PLC_Fail.AlmInputState) ,TGE_Alarm(PLC_Fail,PLC_Fail.AlmInputState) ];
   // Fault Status Bits 11-8 Meaning:
   // 0001= recoverable minor fault
   // 0010 = unrecoverable minor fault
   // 0100 = recoverable major fault
   // 1000 = unrecoverable major fault
   3: [[XIC(mod_status[1].12) ,XIC(mod_status[1].13) ,XIC(mod_status[1].14) ,XIC(mod_status[1].15) ,EQU(mod_faultcode[1],16) ] OTE(SCP_Main_Fail.AlmInputState) ,TGE_Alarm(SCP_Main_Fail,SCP_Main_Fail.AlmInputState) ];
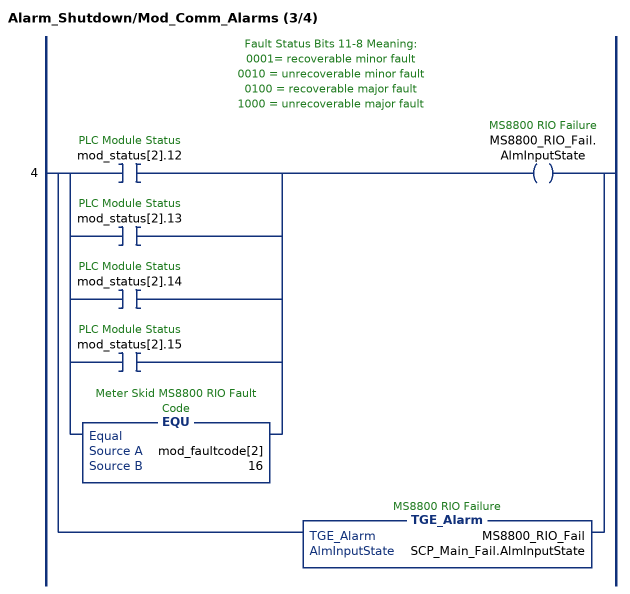
   // Fault Status Bits 11-8 Meaning:
   // 0001= recoverable minor fault
   // 0010 = unrecoverable minor fault
   // 0100 = recoverable major fault
   // 1000 = unrecoverable major fault
   4: [[XIC(mod_status[2].12) ,XIC(mod_status[2].13) ,XIC(mod_status[2].14) ,XIC(mod_status[2].15) ,EQU(mod_faultcode[2],16) ] OTE(MS8800_RIO_Fail.AlmInputState) ,TGE_Alarm(MS8800_RIO_Fail,SCP_Main_Fail.AlmInputState) ];
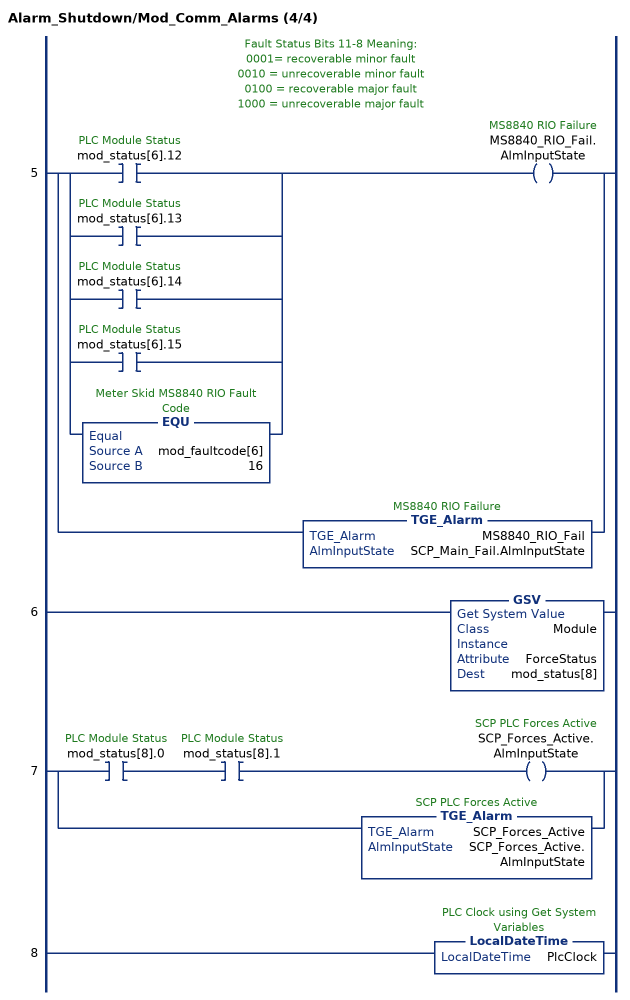
   // Fault Status Bits 11-8 Meaning:
   // 0001= recoverable minor fault
   // 0010 = unrecoverable minor fault
   // 0100 = recoverable major fault
   // 1000 = unrecoverable major fault
   5: [[XIC(mod_status[6].12) ,XIC(mod_status[6].13) ,XIC(mod_status[6].14) ,XIC(mod_status[6].15) ,EQU(mod_faultcode[6],16) ] OTE(MS8840_RIO_Fail.AlmInputState) ,TGE_Alarm(MS8840_RIO_Fail,SCP_Main_Fail.AlmInputState) ];
   6: GSV(Module,,ForceStatus,mod_status[8]);
   7: [XIC(mod_status[8].0) XIC(mod_status[8].1) OTE(SCP_Forces_Active.AlmInputState) ,TGE_Alarm(SCP_Forces_Active,SCP_Forces_Active.AlmInputState) ];
   8: LocalDateTime(PlcClock);
END_ROUTINE

ROUTINE Sta_Alarms   (* ladder *)
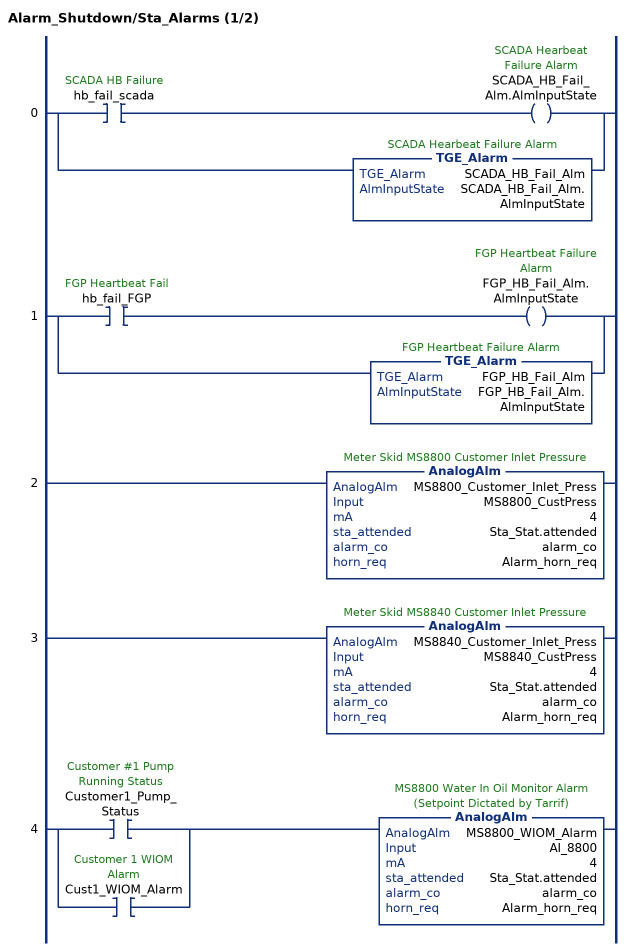
   0: [XIC(hb_fail_scada) OTE(SCADA_HB_Fail_Alm.AlmInputState) ,TGE_Alarm(SCADA_HB_Fail_Alm,SCADA_HB_Fail_Alm.AlmInputState) ];
   1: [XIC(hb_fail_FGP) OTE(FGP_HB_Fail_Alm.AlmInputState) ,TGE_Alarm(FGP_HB_Fail_Alm,FGP_HB_Fail_Alm.AlmInputState) ];
   2: AnalogAlm(MS8800_Customer_Inlet_Press,MS8800_CustPress,4,Sta_Stat.attended,alarm_co,Alarm_horn_req);
   3: AnalogAlm(MS8840_Customer_Inlet_Press,MS8840_CustPress,4,Sta_Stat.attended,alarm_co,Alarm_horn_req);
   4: [XIC(Customer1_Pump_Status) ,XIC(Cust1_WIOM_Alarm) ]AnalogAlm(MS8800_WIOM_Alarm,AI_8800,4,Sta_Stat.attended,alarm_co,Alarm_horn_req);
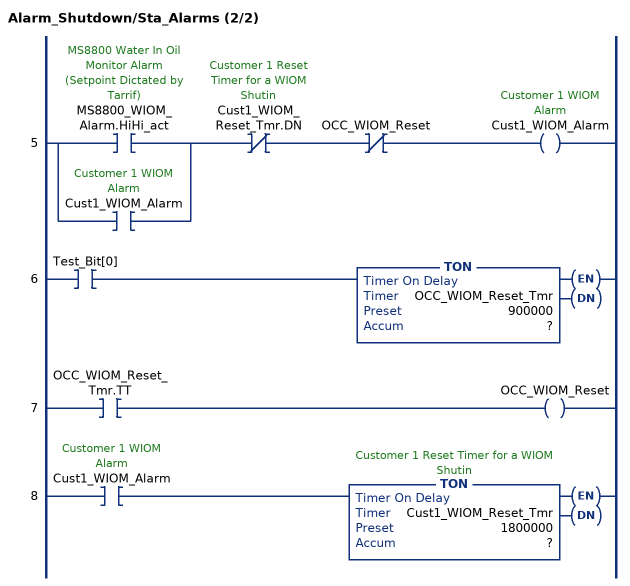
   5: [XIC(MS8800_WIOM_Alarm.HiHi_act) ,XIC(Cust1_WIOM_Alarm) ]XIO(Cust1_WIOM_Reset_Tmr.DN)XIO(OCC_WIOM_Reset)OTE(Cust1_WIOM_Alarm);
   6: XIC(Test_Bit[0])TON(OCC_WIOM_Reset_Tmr,?,?);
   7: XIC(OCC_WIOM_Reset_Tmr.TT)OTE(OCC_WIOM_Reset);
   8: XIC(Cust1_WIOM_Alarm)TON(Cust1_WIOM_Reset_Tmr,?,?);
END_ROUTINE
END_PROGRAM

PROGRAM Auxiliary_Control   (* main routine Main *)

ROUTINE Main   (* ladder *)
END_ROUTINE
END_PROGRAM

PROGRAM Communication   (* main routine Main_Comms *)

ROUTINE EFM_Comms   (* ladder *)
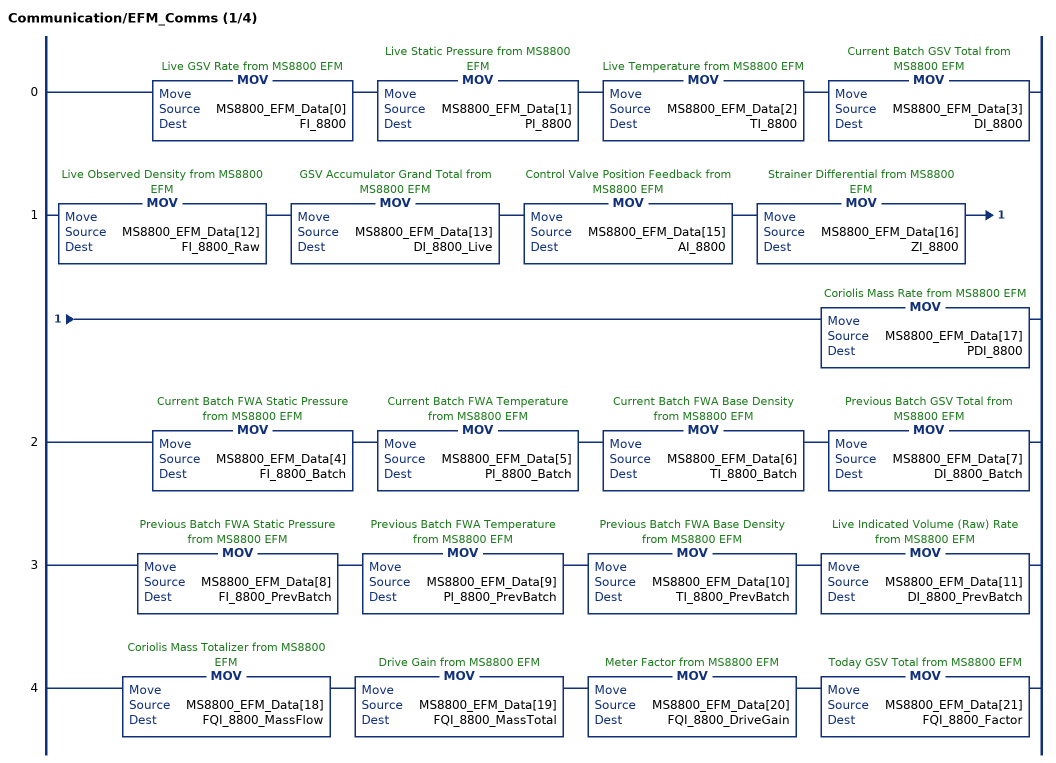
   0: MOV(MS8800_EFM_Data[0],FI_8800)MOV(MS8800_EFM_Data[1],PI_8800)MOV(MS8800_EFM_Data[2],TI_8800)MOV(MS8800_EFM_Data[3],DI_8800);
   1: MOV(MS8800_EFM_Data[12],FI_8800_Raw)MOV(MS8800_EFM_Data[13],DI_8800_Live)MOV(MS8800_EFM_Data[15],AI_8800)MOV(MS8800_EFM_Data[16],ZI_8800)MOV(MS8800_EFM_Data[17],PDI_8800);
   2: MOV(MS8800_EFM_Data[4],FI_8800_Batch)MOV(MS8800_EFM_Data[5],PI_8800_Batch)MOV(MS8800_EFM_Data[6],TI_8800_Batch)MOV(MS8800_EFM_Data[7],DI_8800_Batch);
   3: MOV(MS8800_EFM_Data[8],FI_8800_PrevBatch)MOV(MS8800_EFM_Data[9],PI_8800_PrevBatch)MOV(MS8800_EFM_Data[10],TI_8800_PrevBatch)MOV(MS8800_EFM_Data[11],DI_8800_PrevBatch);
   4: MOV(MS8800_EFM_Data[18],FQI_8800_MassFlow)MOV(MS8800_EFM_Data[19],FQI_8800_MassTotal)MOV(MS8800_EFM_Data[20],FQI_8800_DriveGain)MOV(MS8800_EFM_Data[21],FQI_8800_Factor);
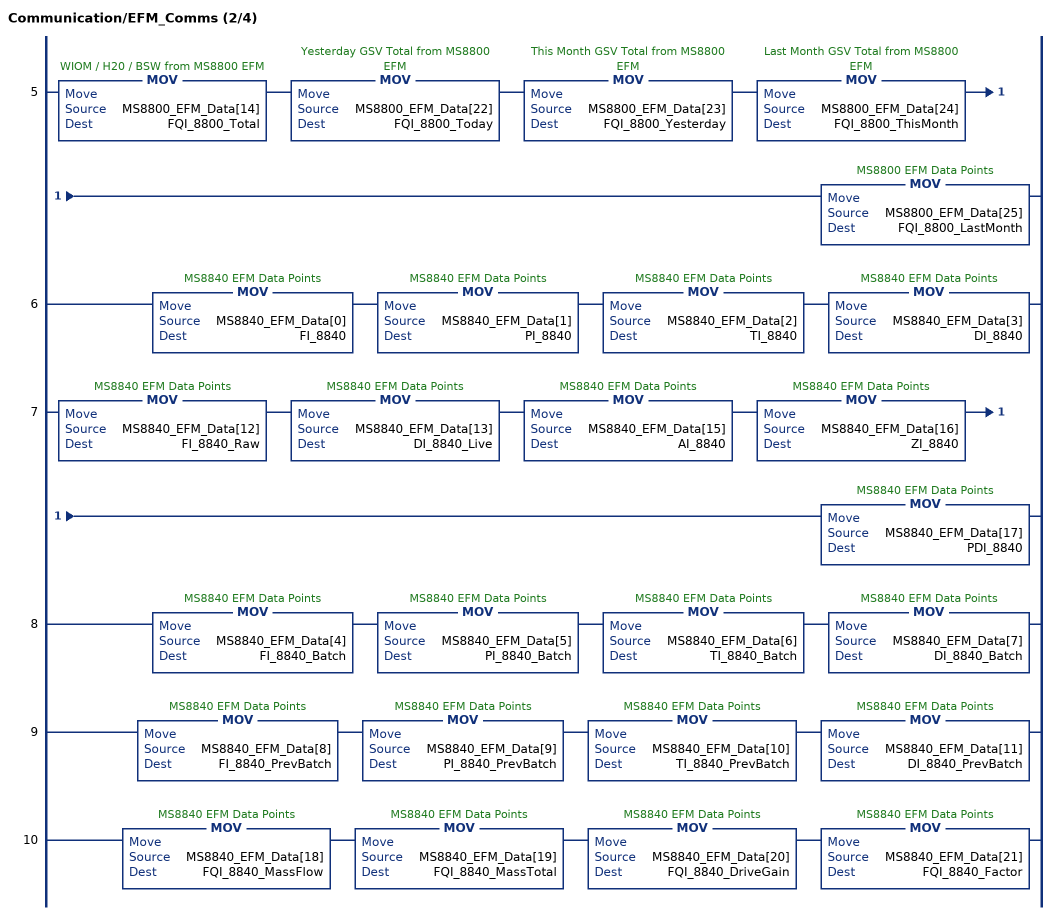
   5: MOV(MS8800_EFM_Data[14],FQI_8800_Total)MOV(MS8800_EFM_Data[22],FQI_8800_Today)MOV(MS8800_EFM_Data[23],FQI_8800_Yesterday)MOV(MS8800_EFM_Data[24],FQI_8800_ThisMonth)MOV(MS8800_EFM_Data[25],FQI_8800_LastMonth);
   6: MOV(MS8840_EFM_Data[0],FI_8840)MOV(MS8840_EFM_Data[1],PI_8840)MOV(MS8840_EFM_Data[2],TI_8840)MOV(MS8840_EFM_Data[3],DI_8840);
   7: MOV(MS8840_EFM_Data[12],FI_8840_Raw)MOV(MS8840_EFM_Data[13],DI_8840_Live)MOV(MS8840_EFM_Data[15],AI_8840)MOV(MS8840_EFM_Data[16],ZI_8840)MOV(MS8840_EFM_Data[17],PDI_8840);
   8: MOV(MS8840_EFM_Data[4],FI_8840_Batch)MOV(MS8840_EFM_Data[5],PI_8840_Batch)MOV(MS8840_EFM_Data[6],TI_8840_Batch)MOV(MS8840_EFM_Data[7],DI_8840_Batch);
   9: MOV(MS8840_EFM_Data[8],FI_8840_PrevBatch)MOV(MS8840_EFM_Data[9],PI_8840_PrevBatch)MOV(MS8840_EFM_Data[10],TI_8840_PrevBatch)MOV(MS8840_EFM_Data[11],DI_8840_PrevBatch);
   10: MOV(MS8840_EFM_Data[18],FQI_8840_MassFlow)MOV(MS8840_EFM_Data[19],FQI_8840_MassTotal)MOV(MS8840_EFM_Data[20],FQI_8840_DriveGain)MOV(MS8840_EFM_Data[21],FQI_8840_Factor);
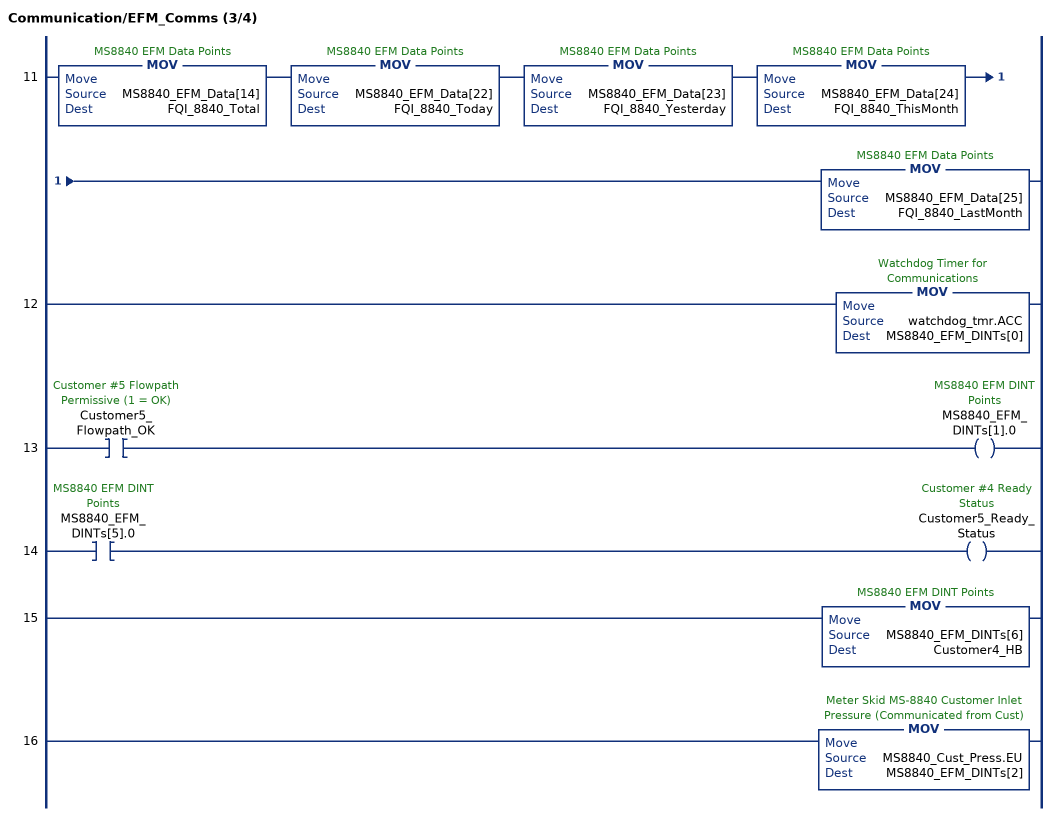
   11: MOV(MS8840_EFM_Data[14],FQI_8840_Total)MOV(MS8840_EFM_Data[22],FQI_8840_Today)MOV(MS8840_EFM_Data[23],FQI_8840_Yesterday)MOV(MS8840_EFM_Data[24],FQI_8840_ThisMonth)MOV(MS8840_EFM_Data[25],FQI_8840_LastMonth);
   12: MOV(watchdog_tmr.ACC,MS8840_EFM_DINTs[0]);
   13: XIC(Customer5_Flowpath_OK)OTE(MS8840_EFM_DINTs[1].0);
   14: XIC(MS8840_EFM_DINTs[5].0)OTE(Customer5_Ready_Status);
   15: MOV(MS8840_EFM_DINTs[6],Customer4_HB);
   16: MOV(MS8840_Cust_Press.EU,MS8840_EFM_DINTs[2]);
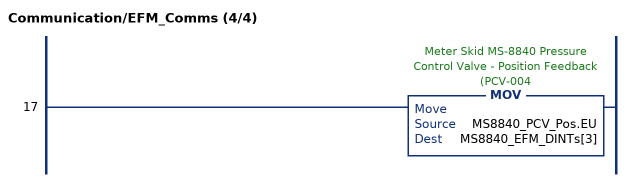
   17: MOV(MS8840_PCV_Pos.EU,MS8840_EFM_DINTs[3]);
END_ROUTINE

ROUTINE FGP_Comms   (* ladder *)
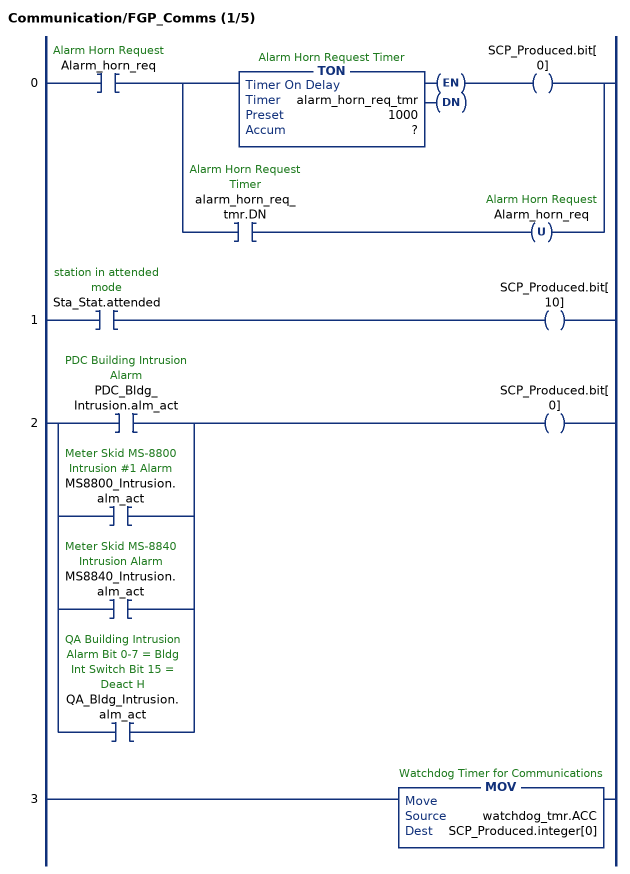
   0: XIC(Alarm_horn_req)[TON(alarm_horn_req_tmr,?,?) OTE(SCP_Produced.bit[0]) ,XIC(alarm_horn_req_tmr.DN) OTU(Alarm_horn_req) ];
   1: XIC(Sta_Stat.attended)OTE(SCP_Produced.bit[10]);
   2: [XIC(PDC_Bldg_Intrusion.alm_act) ,XIC(MS8800_Intrusion.alm_act) ,XIC(MS8840_Intrusion.alm_act) ,XIC(QA_Bldg_Intrusion.alm_act) ]OTE(SCP_Produced.bit[0]);
   3: MOV(watchdog_tmr.ACC,SCP_Produced.integer[0]);
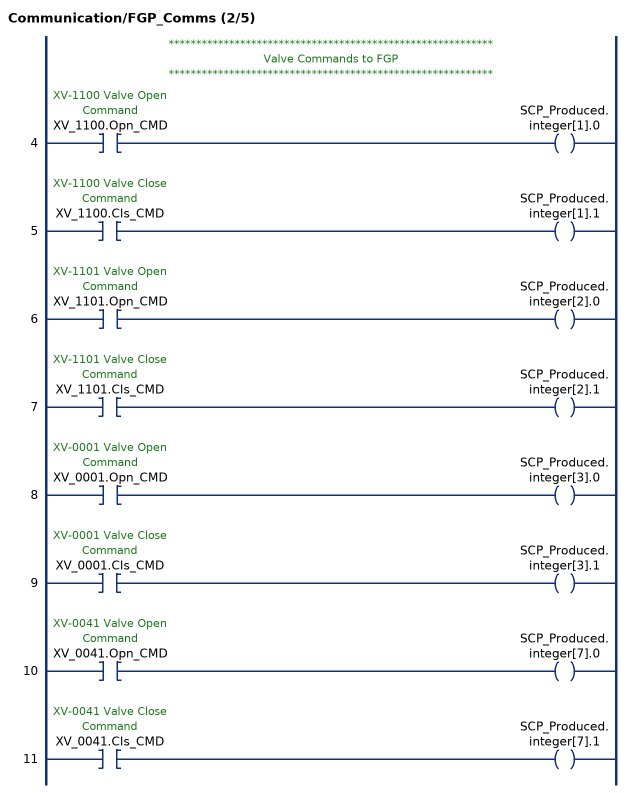
   // ***********************************************************
   // Valve Commands to FGP
   // ***********************************************************
   4: XIC(XV_1100.Opn_CMD)OTE(SCP_Produced.integer[1].0);
   5: XIC(XV_1100.Cls_CMD)OTE(SCP_Produced.integer[1].1);
   6: XIC(XV_1101.Opn_CMD)OTE(SCP_Produced.integer[2].0);
   7: XIC(XV_1101.Cls_CMD)OTE(SCP_Produced.integer[2].1);
   8: XIC(XV_0001.Opn_CMD)OTE(SCP_Produced.integer[3].0);
   9: XIC(XV_0001.Cls_CMD)OTE(SCP_Produced.integer[3].1);
   10: XIC(XV_0041.Opn_CMD)OTE(SCP_Produced.integer[7].0);
   11: XIC(XV_0041.Cls_CMD)OTE(SCP_Produced.integer[7].1);
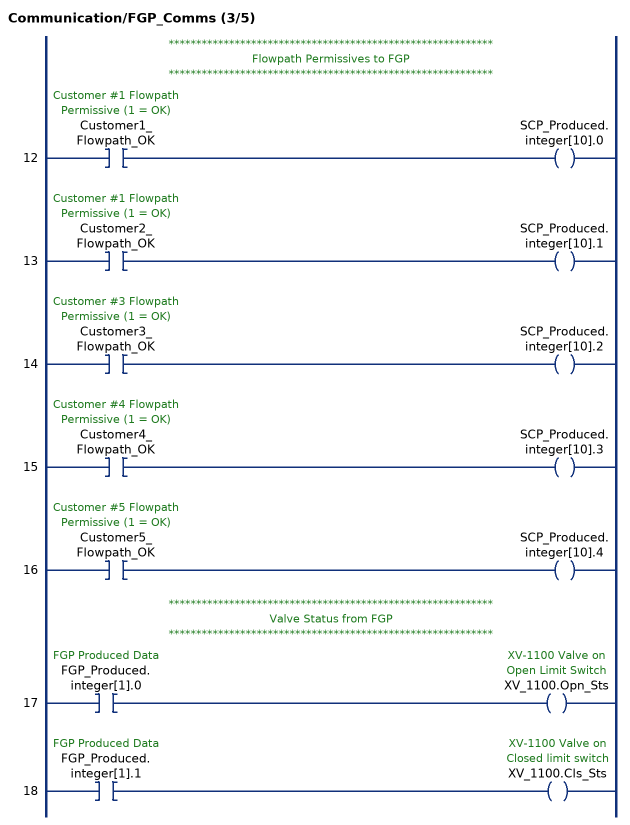
   // ***********************************************************
   // Flowpath Permissives to FGP
   // ***********************************************************
   12: XIC(Customer1_Flowpath_OK)OTE(SCP_Produced.integer[10].0);
   13: XIC(Customer2_Flowpath_OK)OTE(SCP_Produced.integer[10].1);
   14: XIC(Customer3_Flowpath_OK)OTE(SCP_Produced.integer[10].2);
   15: XIC(Customer4_Flowpath_OK)OTE(SCP_Produced.integer[10].3);
   16: XIC(Customer5_Flowpath_OK)OTE(SCP_Produced.integer[10].4);
   // ***********************************************************
   // Valve Status from FGP
   // ***********************************************************
   17: XIC(FGP_Produced.integer[1].0)OTE(XV_1100.Opn_Sts);
   18: XIC(FGP_Produced.integer[1].1)OTE(XV_1100.Cls_Sts);
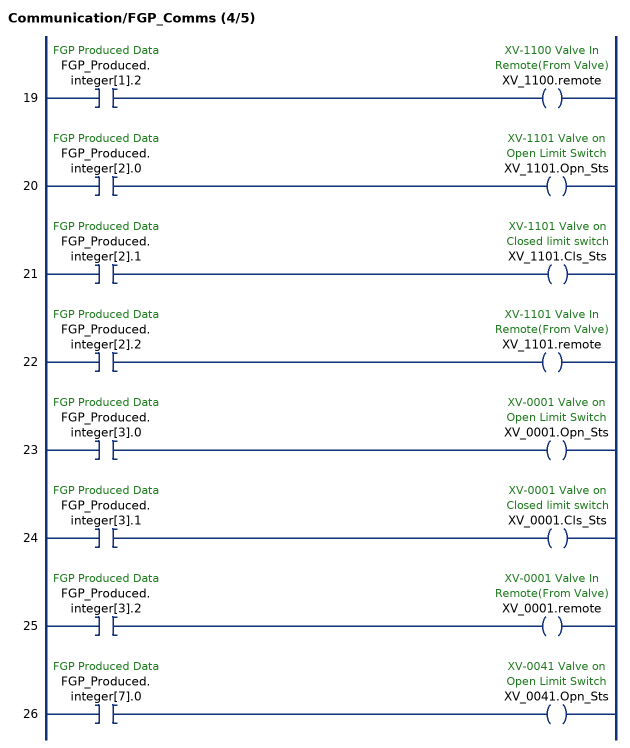
   19: XIC(FGP_Produced.integer[1].2)OTE(XV_1100.remote);
   20: XIC(FGP_Produced.integer[2].0)OTE(XV_1101.Opn_Sts);
   21: XIC(FGP_Produced.integer[2].1)OTE(XV_1101.Cls_Sts);
   22: XIC(FGP_Produced.integer[2].2)OTE(XV_1101.remote);
   23: XIC(FGP_Produced.integer[3].0)OTE(XV_0001.Opn_Sts);
   24: XIC(FGP_Produced.integer[3].1)OTE(XV_0001.Cls_Sts);
   25: XIC(FGP_Produced.integer[3].2)OTE(XV_0001.remote);
   26: XIC(FGP_Produced.integer[7].0)OTE(XV_0041.Opn_Sts);
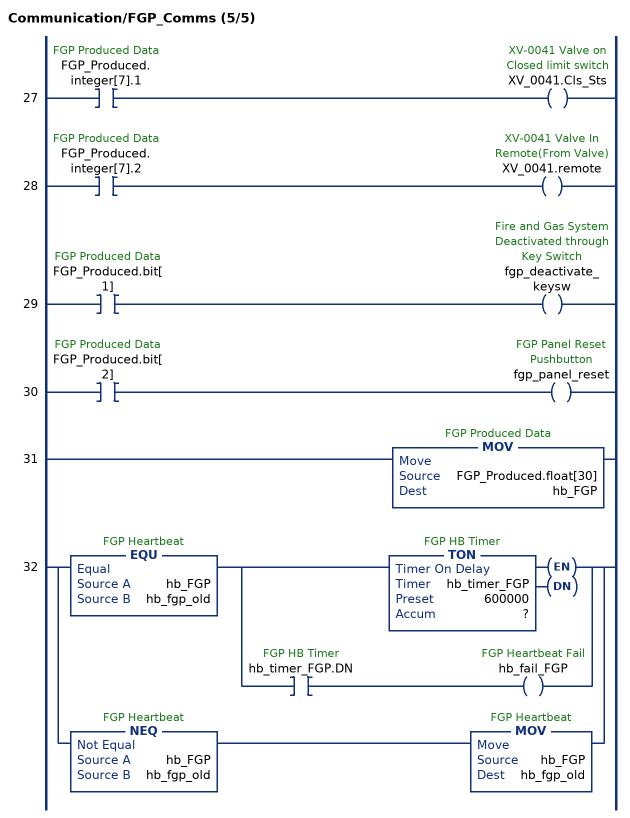
   27: XIC(FGP_Produced.integer[7].1)OTE(XV_0041.Cls_Sts);
   28: XIC(FGP_Produced.integer[7].2)OTE(XV_0041.remote);
   29: XIC(FGP_Produced.bit[1])OTE(fgp_deactivate_keysw);
   30: XIC(FGP_Produced.bit[2])OTE(fgp_panel_reset);
   31: MOV(FGP_Produced.float[30],hb_FGP);
   32: [EQU(hb_FGP,hb_fgp_old) [TON(hb_timer_FGP,?,?) ,XIC(hb_timer_FGP.DN) OTE(hb_fail_FGP) ] ,NEQ(hb_FGP,hb_fgp_old) MOV(hb_FGP,hb_fgp_old) ];
END_ROUTINE

ROUTINE Hereford_Comms   (* ladder *)
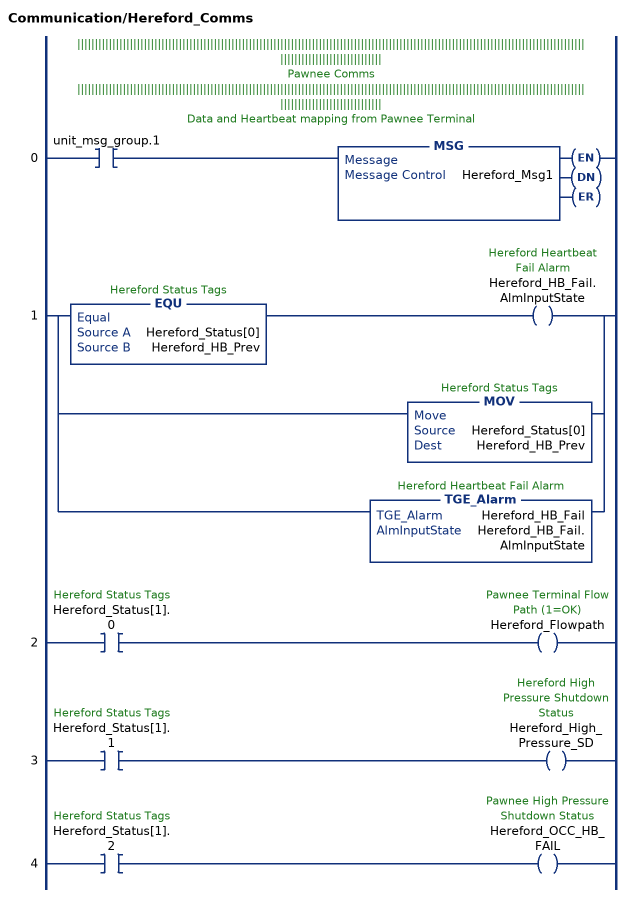
   // ||||||||||||||||||||||||||||||||||||||||||||||||||||||||||||||||||||||||||||||||||||||||||||||||||||||||||||||||||||||||||||||||||||||||||||||||||||||||||||||||||||||||||||||
   // Pawnee Comms
   // ||||||||||||||||||||||||||||||||||||||||||||||||||||||||||||||||||||||||||||||||||||||||||||||||||||||||||||||||||||||||||||||||||||||||||||||||||||||||||||||||||||||||||||||
   // Data and Heartbeat mapping from Pawnee Terminal
   0: XIC(unit_msg_group.1)MSG(Hereford_Msg1);
   1: [EQU(Hereford_Status[0],Hereford_HB_Prev) OTE(Hereford_HB_Fail.AlmInputState) ,MOV(Hereford_Status[0],Hereford_HB_Prev) ,TGE_Alarm(Hereford_HB_Fail,Hereford_HB_Fail.AlmInputState) ];
   2: XIC(Hereford_Status[1].0)OTE(Hereford_Flowpath);
   3: XIC(Hereford_Status[1].1)OTE(Hereford_High_Pressure_SD);
   4: XIC(Hereford_Status[1].2)OTE(Hereford_OCC_HB_FAIL);
END_ROUTINE
